# EPICS autosave request: optics/opticsApp/Db/MLLH_soft_settings.req
$(P)$(Q)xLen
$(P)$(Q)zNoseLen
$(P)$(Q)zBendLen
file basic_motor_settings.req P=$(P),Q=$(Q),M=$(Q)th
file basic_motor_settings.req P=$(P),Q=$(Q),M=$(Q)z
file basic_motor_settings.req P=$(P),Q=$(Q),M=$(Q)x
